// SIMATIC S7-200 SMART project (STEP 7-Micro/WIN SMART), CPU SR40

SYMBOL_TABLE 系统符号
Always_On        SM0.0    // 始终接通
First_Scan_On    SM0.1    // 仅在第一个扫描周期时接通
END_SYMBOL_TABLE

ORGANIZATION_BLOCK MAIN:OB1
TITLE=程序注释
BEGIN
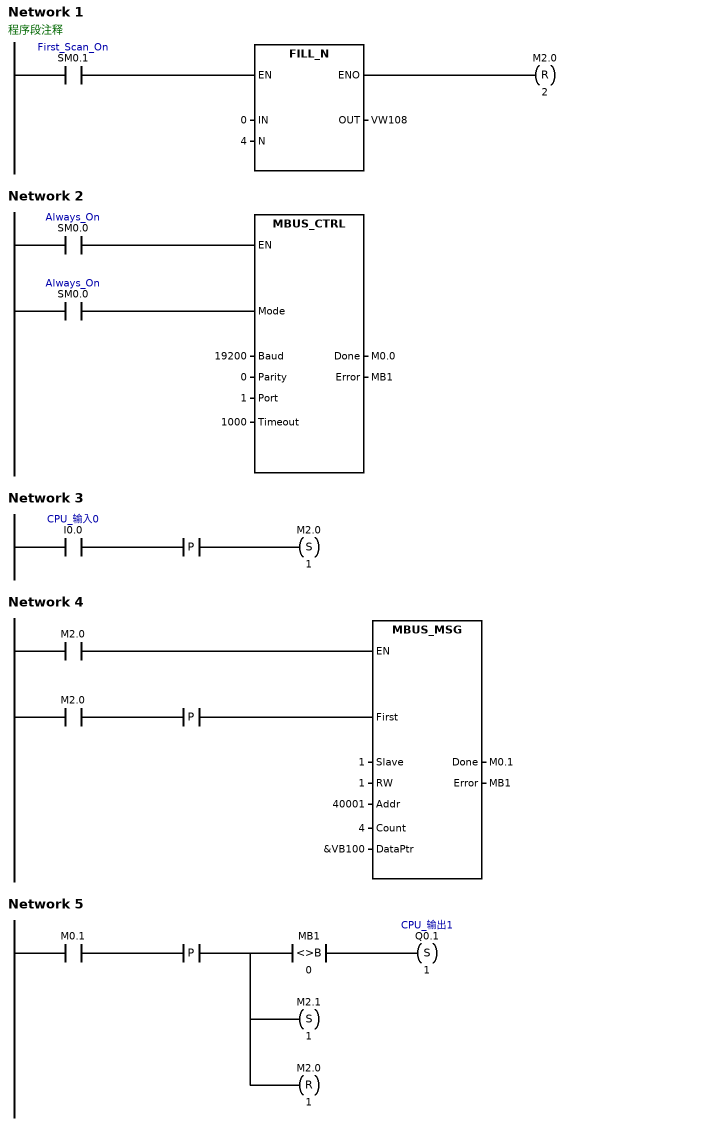
Network 1
// 程序段注释
LD     First_Scan_On:SM0.1
FILL   0, VW108, 4
AENO
R      M2.0, 2
Network 2
LD     Always_On:SM0.0
=      L60.0
LD     Always_On:SM0.0
=      L63.7
LD     L60.0
CALL   MBUS_CTRL:SBR1, L63.7, 19200, 0, 1, 1000, M0.0, MB1
Network 3
LD     CPU_输入0:I0.0
EU
S      M2.0, 1
Network 4
LD     M2.0
=      L60.0
LD     M2.0
EU
=      L63.7
LD     L60.0
CALL   MBUS_MSG:SBR2, L63.7, 1, 1, 40001, 4, &VB100, M0.1, MB1
Network 5
LD     M0.1
EU
LPS
AB<>   MB1, 0
S      CPU_输出1:Q0.1, 1
LRD
S      M2.1, 1
LPP
R      M2.0, 1
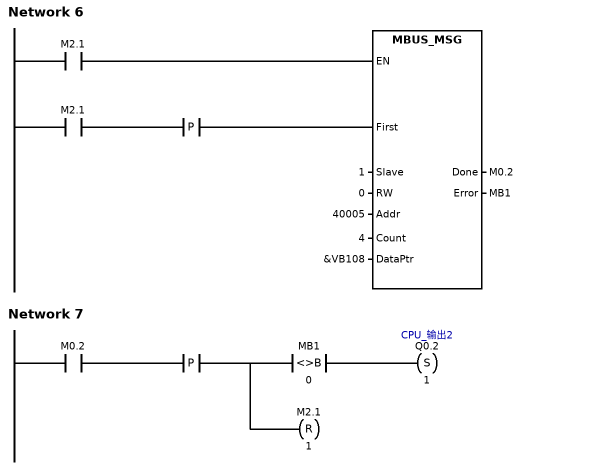
Network 6
LD     M2.1
=      L60.0
LD     M2.1
EU
=      L63.7
LD     L60.0
CALL   MBUS_MSG:SBR2, L63.7, 1, 0, 40005, 4, &VB108, M0.2, MB1
Network 7
LD     M0.2
EU
LPS
AB<>   MB1, 0
S      CPU_输出2:Q0.2, 1
LPP
R      M2.1, 1
END_ORGANIZATION_BLOCK

// SBR1: protected block, not included

// SBR2: protected block, not included

// SBR3: protected block, not included
